// TIA Portal V17 export
// export: Created 2022-07-20T07:02:32.6949632Z, ExportSetting WithDefaults, DisplayName Totally Integrated Automation Portal, DisplayVersion V17, DisplayName TIA Portal Openness, DisplayVersion V17, DisplayName TIA Portal Version Control Interface, DisplayVersion V17, DisplayName SINAMICS Startdrive Advanced, DisplayVersion V17, DisplayName SINAMICS Startdrive G130, G150, S120, S150, SINAMICS MV, S210, DisplayVersion V17, DisplayName SINAMICS Startdrive G110M, G120, G120C, G120D, G120P, G115D, DisplayVersion V17, DisplayName STEP 7 Professional, DisplayVersion V17, DisplayName STEP 7 Safety, DisplayVersion V17, DisplayName WinCC Advanced, DisplayVersion V17
FUNCTION_BLOCK "FB11010_Power"   // FB11010, LAD
{ S7_Optimized_Access := 'TRUE' }
VERSION : 0.1
// stored: AutoNumber false, IsIECCheckEnabled false, IsRetainMemResEnabled false, MemoryReserve 100, SetENOAutomatically false, UDAEnableTagReadback false
   VAR_INPUT
      ActualState : "stStandardMgiOmacStatesBool";
   END_VAR
   VAR_OUTPUT
      EnbaleHeating : Bool;
      MainPower1 : Bool;
      MainPower2 : Bool;
   END_VAR
BEGIN

REGION Network 1 (SCL): Output management
   IF #ActualState.Clearing THEN
       #EnbaleHeating := TRUE;
       #MainPower1 := TRUE;
       #MainPower2 := TRUE;
   END_IF;

   IF #ActualState.Aborting THEN
       #EnbaleHeating := FALSE;
       #MainPower1 := FALSE;
       #MainPower2 := FALSE;
   END_IF;
END_REGION
END_FUNCTION_BLOCK
